TYPE HMISettingLineInterface :
STRUCT
	CaptionSettingLine	:	STRING;
	VisibilitySettingLine	:	BOOL;
	SettingLineButtons	:	ARRAY[1..3] OF HMIButtonSettingLineInterface;
END_STRUCT
END_TYPE

(* stored: Version 1.1.0.1
   DUT HMISettingLineInterface: Id {a4fd7520-d467-4c44-a00c-1450f8a2c779} *)
